{attribute 'qualified_only'}
VAR_GLOBAL
	Morning 		: BOOL	 ;
	
	WakeUp			: BOOL	 ;
	DateCheck		: BOOL	 ;
	ComeBackHome	: BOOL	 ;
	TakeShower		: BOOL	 ;
	GoToBed			: BOOL 	 ;
	MakeTheBed		: BOOL   ;
	MakeCoffee		: BOOL	 ;
	EatBreakfast	: BOOL	 ;
	
			
END_VAR

(* stored: Version 1.1.0.1, ProductVersion 3.1.4024.12
   GVL GVL: Id {0eb15bf5-694d-4967-b4b9-b366a288d4ce} *)
